FUNCTION_BLOCK FB_AuxiliaryPump
VAR_IN_OUT
	AuxiliaryPump : ST_AuxiliaryPump;
END_VAR
VAR_INPUT
	Turbo : ST_AgilentPTM;	
END_VAR
VAR
	TOFtmr : TOF;
END_VAR

TOFtmr(IN := Turbo.i_xR1 OR Turbo.i_xSTART, PT := T#150S );
AuxiliaryPump.q_ContactClosed :=AuxiliaryPump.i_xRunSW OR TOFtmr.q;

END_FUNCTION_BLOCK

(* stored: Version 1.1.0.1, ProductVersion 3.1.4020.12
   POU FB_AuxiliaryPump: Id {997755b9-52a8-4f6d-a9f1-2dbeec2b934b}, SpecialFunc None *)
